(* IEC 61131-3 sources: CodesysTest/alpha/export/Pro18_1174_04.dev/Plc Logic/Application/Motors/Applied Motion/FB_AppliedMotionBagDeliveryMotor.pou, 2 files *)

(* ---- FB_AppliedMotionBagDeliveryMotor.pou.st ---- *)
(*#-#-#-#-#-#-#-#-#-#---Declaration---#-#-#-#-#-#-#-#-#-#-#-#-#*)

FUNCTION_BLOCK FB_AppliedMotionBagDeliveryMotor EXTENDS FB_AppliedMotionStepServoTCP
VAR_INPUT
END_VAR
VAR_OUTPUT
END_VAR
VAR
    sendParameters : FB_SendUserRegistersAppliedMotionTCP();
    sendBagMoveCommand : FB_SendBagMoveAppliedMotionTCP();
END_VAR
(*#-#-#-#-#-#-#-#-#-#---Implementation---#-#-#-#-#-#-#-#-#-#-#-#-#*)

sendMoveCommand(Slave := slave);
sendBagMoveCommand(Slave := slave);
sendOpcodeCommand(Slave := slave);
sendParameters(Slave := slave);

commandSuccessful S= ((sendMoveCommand.xDone OR sendOpcodeCommand.xDone OR sendBagMoveCommand.xDone) AND NOT status.inPosition) OR sendParameters.xDone;

(* ---- MoveDistanceFinal.m.st ---- *)
(*#-#-#-#-#-#-#-#-#-#---Declaration---#-#-#-#-#-#-#-#-#-#-#-#-#*)

METHOD MoveDistanceFinal
VAR_INPUT
    distance : REAL;        //Distance to move in inches
    acceleration : INT;        //Acceleration in RPM/sec
    deceleration : INT;        //Deceleration in RPM/sec
    velocity : INT;            //Velocity in .25RPM
END_VAR
(*#-#-#-#-#-#-#-#-#-#---Implementation---#-#-#-#-#-#-#-#-#-#-#-#-#*)

distanceToMoveInSteps.rawValue := REAL_TO_DINT((distance) * stepsPerInchSetpoint);
IF reversePolarity THEN
    distanceToMoveInSteps.rawValue := distanceToMoveInSteps.rawValue * -1;
END_IF
commandSuccessful := FALSE;
ModbusLongHandler.Unpack(distanceToMoveInSteps);
sendBagMoveCommand.acceleration := acceleration;
sendBagMoveCommand.deceleration := deceleration;
sendBagMoveCommand.velocity := velocity;
sendBagMoveCommand.distanceHighWord := distanceToMoveInSteps.highWord;
sendBagMoveCommand.distanceLowWord := distanceToMoveInSteps.lowWord;
sendBagMoveCommand.opcode := STEP_SERVO_OPCODES.QUEUE_LOAD_AND_EXECUTE;
sendBagMoveCommand.programToRun := 2;
sendBagMoveCommand.Execute();
